PROGRAM pouS2Alarms
VAR
	idbMsgAlarm: FB_CheckMessageBounds;

END_VAR

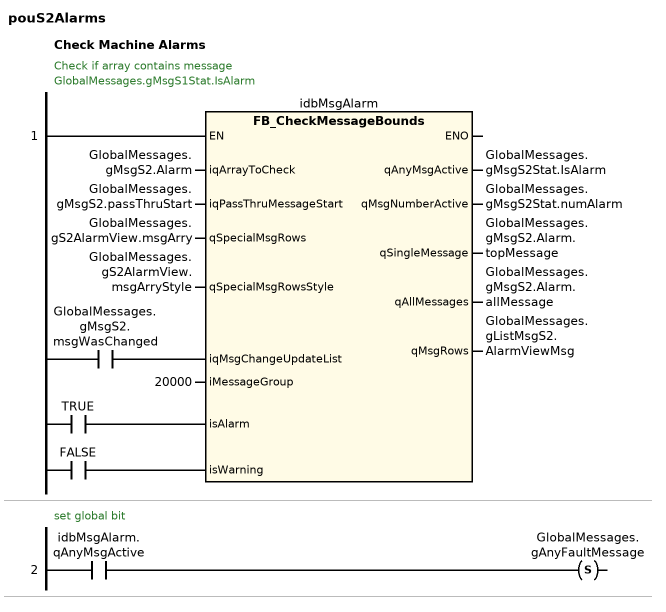
// NETWORK 1: Check Machine Alarms
// Check if array contains message
//
// GlobalMessages.gMsgS1Stat.IsAlarm
idbMsgAlarm(
    iqArrayToCheck := GlobalMessages.gMsgS2.Alarm,
    iqPassThruMessageStart := GlobalMessages.gMsgS2.passThruStart,
    qSpecialMsgRows := GlobalMessages.gS2AlarmView.msgArry,
    qSpecialMsgRowsStyle := GlobalMessages.gS2AlarmView.msgArryStyle,
    iqMsgChangeUpdateList := GlobalMessages.gMsgS2.msgWasChanged,
    iMessageGroup := 20000,
    isAlarm := TRUE,
    isWarning := FALSE,
    qAnyMsgActive => GlobalMessages.gMsgS2Stat.IsAlarm,
    qMsgNumberActive => GlobalMessages.gMsgS2Stat.numAlarm,
    qSingleMessage => GlobalMessages.gMsgS2.Alarm.topMessage,
    qAllMessages => GlobalMessages.gMsgS2.Alarm.allMessage,
    qMsgRows => GlobalMessages.gListMsgS2.AlarmViewMsg); // FB_CheckMessageBounds

// NETWORK 2
// set global bit
GlobalMessages.gAnyFaultMessage S= idbMsgAlarm.qAnyMsgActive;

END_PROGRAM

(* stored: Version 1.1.0.1, ProductVersion 3.1.4024.12
   POU pouS2Alarms: Id {fbc2ad47-b03b-4448-bd52-7d18a39f8fe2}, SpecialFunc None *)
